// TwinCAT 3 PLC project HMI
// ProgramVersion: 3.1.4023.0
// libraries:
//   Tc2_Standard, * (Beckhoff Automation GmbH)
//   Tc2_System, * (Beckhoff Automation GmbH)
//   Tc2_Utilities, * (Beckhoff Automation GmbH)
//   Tc3_Database, * (Beckhoff Automation GmbH)
//   Tc3_Module, * (Beckhoff Automation GmbH)
// project tree:
//   DUTs/Bundle and Material/ BasicBundle.TcDUT, Bundle.TcDUT, Interval.TcDUT, Material.TcDUT, PositionMaterials.TcDUT
//   DUTs/Enums/ DatabaseStep.TcDUT, MaterialType.TcDUT
//   DUTs/ FB_TcpBlock.TcPOU, ST_TcpStructure.TcDUT
//   DUTs/String Builder/ StringBuilder.TcPOU
//   GVLs/ GVL.TcGVL
//   / PlcTask.TcTTO
//   POUs/Helper Functions/ GetMasterLength.TcPOU, GetMaterialLength.TcPOU, IntervalIsvalid.TcPOU, MetricMaterialDimensions.TcPOU, PositionIsValid.TcPOU
//   POUs/ MAIN.TcPOU, FindBundlesFromDB.TcPOU, RecalibrateRecipe.TcPOU, SqlDbReadWrite.TcPOU
// (motion and I/O tree: see PLC project dispatch)
// real-time tasks:
//   TASK PlcTask: cycle T#10ms, priority 20, ADS port 350
//   TASK PlcTask1: cycle T#10ms, priority 21, ADS port 351

CONFIGURATION HMI
    RESOURCE PLC ON TwinCAT3
        TASK PlcTask(INTERVAL := T#10ms, PRIORITY := 21);
        PROGRAM MAIN WITH PlcTask : MAIN;
    END_RESOURCE
END_CONFIGURATION

// ---- DUTs/Bundle and Material/BasicBundle.TcDUT
TYPE BasicBundle :
STRUCT
	id : STRING;
	
	weight : REAL;
	
	length : USINT;
	width : USINT;
	height : USINT;
	
	extrusionWeight : REAL;
	extrusionWidth : USINT;
	extrusionHeight : USINT;
	
	pieces : USINT;
	layers : USINT;
	piecesPerLayer : USINT;
END_STRUCT
END_TYPE

(*
barebones structure for essential bundle data that can be displayed on the HMI
refer to full structure for full recipe
*)

// ---- DUTs/Bundle and Material/Bundle.TcDUT
{attribute 'enable_dynamic_creation'}
TYPE Bundle :
STRUCT
	id : STRING;
	
	weight : REAL;
	length : USINT;
	width : USINT;
	height : USINT;
	
	pieces : USINT;
	layers : USINT;
	piecesPerLayer : USINT;
	
	extrusionWeight : REAL;
	extrusionHeight : USINT;
	extrusionWidth : USINT;
	
	processes : (AUTO_RE, AUTO_SS, MAN_RE, MAN_SS);
	reqProcesses : ARRAY[0..3] OF BOOL;
	
	coverPaper : ARRAY[0..1] OF BOOL;
	coverCardboard : ARRAY[0..1] OF BOOL;
	
	paperTop : ARRAY[0..GVL.maxPairs] OF Interval;
	paperLeft : ARRAY[0..GVL.maxPairs] OF Interval;
	paperRight : ARRAY[0..GVL.maxPairs] OF Interval;
	paperBottom : ARRAY[0..GVL.maxPairs] OF Interval;
		
	cardboard : ARRAY[0..GVL.maxPairs] OF PositionMaterials;
	cornerGuard : ARRAY[0..GVL.maxPairs] OF PositionMaterials;
	
	combinedCardboardCornerGuard : ARRAY[0..(GVL.maxPairs*2)] OF PositionMaterials;
	
	chipboard : ARRAY[0..GVL.maxPairs] OF PositionMaterials;
	woodBunk : ARRAY[0..GVL.maxPairs] OF PositionMaterials;
	
	cardboard_over_cornerGuard : BOOL;
	
	currStep : USINT; //for runtime use only
	
	//for production log database
	timeStart : TIMESTRUCT;
	timeDone : TIMESTRUCT;
END_STRUCT
END_TYPE

// ---- DUTs/Bundle and Material/Interval.TcDUT
TYPE Interval :
STRUCT
	startPos : REAL;
	endPos : REAL;
END_STRUCT
END_TYPE

// ---- DUTs/Bundle and Material/Material.TcDUT
TYPE Material :
STRUCT
	code : STRING;
	width : REAL;
	length : REAL;
	
	widthMM : INT;
	lengthMM : INT;
END_STRUCT
END_TYPE
(*
use this struct to keep track of where materials are
materials enter the system when pulled from their magazine/skid and exit the system when placed on the bundle or otherwise lost
*)

// ---- DUTs/Bundle and Material/PositionMaterials.TcDUT
TYPE PositionMaterials :
STRUCT
	position : REAL := GVL.nullPos; //default value is set to predefined constant if bundle needs less than 32 position material pairs
	
	top : STRING;
	left : STRING;
	right : STRING;
	bottom : STRING;
	
	topLeft : STRING;
	topLeftFold : USINT;
	
	topRight : STRING;
	topRightFold : USINT;
	
	bottomLeft : STRING;
	bottomLeftFold : USINT;
	
	bottomRight : STRING;
	bottomRightFold : USINT;

	wrapPoints : USINT;
	wrapRotations : USINT;
END_STRUCT
END_TYPE

// ---- DUTs/Enums/DatabaseStep.TcDUT
{attribute 'qualified_only'}
{attribute 'strict'}
TYPE DatabaseStep :
(
	RESET,
	DISCONNECT, 
	CONNECT, 
	IDLE, 
	EXECUTE, 
	LOAD_DATA,
	
	size
);
END_TYPE

// ---- DUTs/Enums/MaterialType.TcDUT
{attribute 'qualified_only'}
{attribute 'strict'}
{attribute 'to_string'}
TYPE MaterialType :
(
	PAPER,
	CARDBOARD,
	CORNER_GUARD,
	CHIPBOARD,
	WOOD_BUNK
);
END_TYPE

// ---- DUTs/ST_TcpStructure.TcDUT
TYPE ST_TcpStructure :
STRUCT
	transmissionTime : TIMESTRUCT;
	dataType : (NO_DATA, BUNDLE_TRANSFER, BUNDLE_ETA, GENERAL_EVENT)INT;
	timestamp : TIMESTRUCT;
	binaryData : ARRAY[0..50000] OF BYTE;
	jsonData : STRING(2000);
	xmlData : STRING(2000);
END_STRUCT
END_TYPE

// ---- GVLs/GVL.TcGVL
{attribute 'qualified_only'}
VAR_GLOBAL CONSTANT
	maxPairs : USINT := 16;
	initArraySize : USINT := 4;
	
	nullPos : REAL := -1;
	
	numMaterials : INT := 32;
	allMaterials : ARRAY[0..numMaterials] OF Material := [
		(code := 'PAP28', width := 28, length := -1),
		
		(code := 'CAR20S', width := 20, length := 30),
		(code := 'CAR20M', width := 20, length := 45),
		(code := 'CAR20L', width := 20, length := 60),
		(code := 'CAR28S', width := 28, length := 30),
		(code := 'CAR28M', width := 28, length := 45),
		(code := 'CAR28L', width := 28, length := 60),
		
		(code := 'COR48', width := 1.5, length := 48),
		(code := 'COR96', width := 1.5, length := 96),
		
		(code := 'CIP18', width := 20, length := 18),
		(code := 'CIP54', width := 20, length := 54),
		
		(code := 'WDT20', width := 20, length := 2.5),
		(code := 'WDT22', width := 22, length := 2.5),
		(code := 'WDT28', width := 28, length := 2.5),
		
		(code := 'WDB20', width := 20, length := 2.5),
		(code := 'WDB22', width := 22, length := 2.5),
		(code := 'WDB28', width := 28, length := 2.5),
		
		(code := 'WDS08', width := 8, length := 2.5),
		(code := 'WDS10', width := 10, length := 2.5),
		(code := 'WDS12', width := 12, length := 2.5),
		(code := 'WDS14', width := 14, length := 2.5),
		(code := 'WDS8x8', width := 16, length := 2.5),
		(code := 'WDS8x10', width := 18, length := 2.5),
		(code := 'WDS20', width := 20, length := 2.5),
		(code := 'WDS22', width := 22, length := 2.5),
		(code := 'WDS12x12', width := 24, length := 2.5),
		(code := 'WDS12x14', width := 26, length := 2.5),
		(code := 'WDS28', width := 28, length := 2.5),
		(code := 'WDS20x10', width := 30, length := 2.5),
		(code := 'WDS20x12', width := 32, length := 2.5),
		
		(code := 'WDW20', width := 20, length := 6),
		(code := 'WDW22', width := 22, length := 6)]; //+1 null material
		
	cipBuffer : INT := 2; //2in or 50mm
END_VAR
VAR_GLOBAL
	AmsNetId : T_AmsNetId;
	systemTime : TIMESTRUCT;
	
	originalBundle : Bundle; //this one stays internal
	confirmedBundle : Bundle; //this oen is editable by the HMI
END_VAR

// ---- POUs/MAIN.TcPOU
PROGRAM MAIN
VAR
	getLocalAmsNetId : FB_GetLocalAmsNetId;
	getLocalSystemTime : FB_LocalSystemTime;
	
	id : STRING;
	queryId : STRING;
	stringBuilder : StringBuilder;
	
	original : Bundle;
	confirmed : Bundle;
END_VAR
VAR CONSTANT
	AUTO_RE : INT := 0;
	AUTO_SS : INT := 1;
	MAN_RE : INT := 2;
	MAN_SS : INT := 3;
END_VAR

getLocalSystemTime(
	sNetID:= GVL.AmsNetId, 
	bEnable:= TRUE, 
	dwCycle:= 1, 
	dwOpt:= , 
	tTimeout:= , 
	bValid=> , 
	systemTime=> GVL.systemTime, 
	tzID=> );

IF NOT setup() THEN
	RETURN;
END_IF

MetricMaterialDimensions(GVL.allMaterials);

queryId := stringBuilder
	.concatWith('%')
	.concatWith(id)
	.concatWith('%')
	.getResult();
stringBuilder.reset();

FindBundlesFromDB(id := queryId);

IF confirmed.length <> original.length THEN
	RecalibrateRecipe(original := original, confirmed := confirmed);
	
	IF RecalibrateRecipe.reject THEN //send to manual processes
		confirmed.reqProcesses[AUTO_RE] := FALSE;
		confirmed.reqProcesses[AUTO_SS] := FALSE;
		confirmed.reqProcesses[MAN_RE] := TRUE;
		confirmed.reqProcesses[MAN_SS] := TRUE;	
	END_IF
ELSE
	//use as is
END_IF

METHOD setup : BOOL
VAR_INPUT
END_VAR
getLocalAmsNetId(
	bExecute:= TRUE, 
	tTimeOut:= T#1S, 
	bBusy=> , 
	bError=> , 
	nErrId=> , 
	AddrString=> GVL.AmsNetId, 
	AddrBytes=> );

getLocalAmsNetId.bExecute := FALSE;

setup := (GVL.AmsNetId <> '' AND GVL.AmsNetId <> '0.0.0.0.0.0');
END_METHOD

END_PROGRAM

// ---- DUTs/String Builder/StringBuilder.TcPOU
FUNCTION_BLOCK StringBuilder
VAR
	result : STRING(1000);
END_VAR

METHOD concatStringArray : STRING(1000)
VAR_IN_OUT
	arr : ARRAY[*] OF STRING;
END_VAR
VAR
	temp : STRING(1000);
END_VAR
END_METHOD

METHOD concatWith : REFERENCE TO StringBuilder
VAR_INPUT
	target : STRING;
END_VAR
CONCAT2(ADR(result), ADR(target), ADR(result), SIZEOF(result));
concatWith REF= THIS^;
END_METHOD

METHOD getResult : STRING(1000)
getResult := result;
END_METHOD

METHOD reset : BOOL
VAR_INPUT
END_VAR
result := '';
END_METHOD

END_FUNCTION_BLOCK

// ---- POUs/Helper Functions/MetricMaterialDimensions.TcPOU
FUNCTION MetricMaterialDimensions : BOOL
VAR_IN_OUT
	materials : ARRAY[*] OF Material;
END_VAR
VAR
	i : DINT;
END_VAR

FOR i:=LOWER_BOUND(materials, 1) TO UPPER_BOUND(materials, 1) BY 1 DO
	materials[i].lengthMM := TO_INT(materials[i].length * 25.4);
	materials[i].widthMM := TO_INT(materials[i].width * 25.4);
END_FOR

END_FUNCTION

// ---- POUs/FindBundlesFromDB.TcPOU
PROGRAM FindBundlesFromDB EXTENDS SqldbReadWrite
VAR_INPUT
	id : STRING;
END_VAR
VAR_OUTPUT
	basicBundlesArr : ARRAY[0..20-1] OF BasicBundle;
END_VAR
VAR
	fbSQLCommand : FB_SQLCommandEvt(sNetID := '', tTimeout := T#5S);
	fbSQLDatabase : FB_SQLDatabaseEvt (sNetID := '', tTimeout := T#5S);
	fbSQLResult : FB_SQLResultEvt(sNetID:='', tTimeout:=T#5S);
	
	query : STRING(1000);
	//step : (RESET, CONNECT, IDLE, EXECUTE, LOAD_DATA, DISCONNECT);
END_VAR
VAR
	stringBuilder : StringBuilder;
	i : INT;
END_VAR

IF NOT ready THEN
	setup();
	RETURN;
END_IF

CASE step OF
	(*
	RESET:
		step := DISCONNECT;
		
	CONNECT:
		IF fbSQLDatabase.Connect(1) THEN
			IF NOT fbSqlDatabase.bError THEN
				step := IDLE;
			END_IF
		END_IF
	*)
	IDLE:
		IF fbSQLDatabase.CreateCmd(ADR(fbSQLCommand)) THEN
			step := EXECUTE;
		END_IF
	
	EXECUTE:
		createQuery();
		IF fbSQLCommand.ExecuteDataReturn(ADR(query), SIZEOF(query), ADR(fbSqlResult)) THEN
			step := IDLE;
		END_IF
	
	LOAD_DATA:
		(*
		fbSqlResult.Read(0, 1, ADR(existingID), SIZEOF(existingID), TRUE, FALSE);
		IF BundleData.id = existingID THEN
			bundleExists := TRUE;
		ELSE
			bundleExists := FALSE;
		END_IF
		IF fbSQLDatabase.Disconnect() THEN
			fbSqlResult.Release();
			checkExistingBundles := TRUE;
			dbCheckStep := CONNECT;
		END_IF
		*)
		
	DISCONNECT:
		IF fbSQLDatabase.Disconnect() THEN
			step := CONNECT;
		END_IF
END_CASE

METHOD PRIVATE createQuery : BOOL
IF id = '' THEN //FINISH WITH OTHER BASIC ATTRIBUTES
	CONCAT2(ADR(query), ADR('SELECT BundleID FROM "Bundle Data - Prototype"'), ADR(query), SIZEOF(query));
ELSE
	CONCAT2(ADR(query), ADR('SELECT BundleID FROM "Bundle Data - Prototype" WHERE BundleID = $''), ADR(query), SIZEOF(query));
	CONCAT2(ADR(query), ADR(id), ADR(query), SIZEOF(query));
	CONCAT2(ADR(query), ADR('$''), ADR(query), SIZEOF(query));
END_IF

createQuery := TRUE;
END_METHOD

METHOD queryBasicAttributes : BOOL
VAR_INPUT
END_VAR
END_METHOD

METHOD queryPackagingRecipe : BOOL
VAR_INPUT
	material : MaterialType;
END_VAR
VAR
	sMaterial : STRING;
END_VAR
sMaterial := TO_STRING(material);

IF i >= GVL.maxPairs THEN
	i := 0;
END_IF

sMaterial := stringBuilder
	.concatWith(
		'SELECT
		(position, top, sides, bottom, upperCorners, upperCorners_foldRatio, lowerCorners, lowerCorners_foldRatio)
		FROM ______ 
		WHERE (')
		
	.concatWith('bundleID = ')
	.concatWith('$'')
	.concatWith(TO_STRING(id))
	.concatWith('$'')
	
	.concatWith(' AND ')
	
	.concatWith('arrayIndex = ')
	.concatWith(TO_STRING(i))
	.concatWith(')')
	.getResult();
(*

FOR i:=0 TO 16 BY 1 DO


select (position, top, sides, bottom, upperCorners, upperCorners_foldRatio, lowerCorners, lowerCorners_foldRatio) from 
where (bundleID = bundle.id and arrayIndex = 1)

//copy the resulting cache into a bundle.<material>[i] (a PositionMaterial struct)
//do this for all material arrays


END_FORR

*)
END_METHOD

METHOD setup : BOOL
CASE step OF
	RESET:
		step := DISCONNECT;
		
	CONNECT:
		IF fbSQLDatabase.Connect(1) THEN
			IF NOT fbSqlDatabase.bError THEN
				step := IDLE;
				setup := TRUE;
			END_IF
		END_IF
		
	DISCONNECT:
		IF fbSQLDatabase.Disconnect() THEN
			step := CONNECT;
		END_IF
END_CASE
END_METHOD

END_PROGRAM

// ---- POUs/SqlDbReadWrite.TcPOU
PROGRAM SqlDbReadWrite
VAR_OUTPUT
	ready : BOOL;
END_VAR
VAR
	fbSQLCommand : FB_SQLCommandEvt(sNetID := '', tTimeout := T#5S);
	fbSQLDatabase : FB_SQLDatabaseEvt (sNetID := '', tTimeout := T#5S);
	fbSQLResult : FB_SQLResultEvt(sNetID:='', tTimeout:=T#5S);
	
	query : STRING(1000);
	step : DatabaseStep;
	
	cachedBuffer : ARRAY[0..100000] OF BYTE;
END_VAR

IF NOT ready THEN
	setup();
	RETURN;
END_IF

CASE step OF
	DatabaseStep.IDLE:
		IF fbSQLDatabase.CreateCmd(ADR(fbSQLCommand)) THEN
			step := DatabaseStep.EXECUTE;
		END_IF
		
	DatabaseStep.EXECUTE:
		IF fbSQLCommand.ExecuteDataReturn(ADR(query), SIZEOF(query), ADR(fbSqlResult)) THEN
			query := '';
			step := DatabaseStep.LOAD_DATA;
		END_IF
		
	DatabaseStep.LOAD_DATA:
		fbSqlResult.Read(
			nStartIndex := 0,
			nRecordCount := 1,
			pData := ADR(cachedBuffer),
			cbData := SIZEOF(cachedBuffer),
			bWithVerifying := FALSE,
			bDataRelease := FALSE);
			
END_CASE

METHOD execute : BOOL
VAR_INPUT
	queryInstruction : STRING(1000);
END_VAR
query := queryInstruction;
END_METHOD

METHOD reset : BOOL
VAR_INPUT
END_VAR
step := RESET;
END_METHOD

METHOD setup : BOOL
CASE step OF
	DatabaseStep.RESET:
		step := DatabaseStep.DISCONNECT;
		
	DatabaseStep.CONNECT:
		IF fbSQLDatabase.Connect(1) THEN
			IF NOT fbSqlDatabase.bError THEN
				step := DatabaseStep.IDLE;
				setup := TRUE;
			END_IF
		END_IF
		
	DatabaseStep.DISCONNECT:
		IF fbSQLDatabase.Disconnect() THEN
			step := DatabaseStep.CONNECT;
		END_IF
END_CASE
END_METHOD

END_PROGRAM

// ---- POUs/RecalibrateRecipe.TcPOU
PROGRAM RecalibrateRecipe
VAR_INPUT
	original : REFERENCE TO Bundle;
	confirmed : REFERENCE TO Bundle;
END_VAR
VAR
	lengthDifference : REAL;
	minAllowableLength : REAL;
	lengthShortenedDifferenceMax : REAL;
	
	lengthDifferenceFactor : REAL;
	
	cipLength : REAL;
	
	i : INT;
END_VAR
VAR_OUTPUT
	reject : BOOL;
END_VAR

//original REF= GVL.originalBundle;
//confirmed REF= GVL.confirmedBundle;

lengthDifference := confirmed.length - original.length;
minAllowableLength := cipLength + (2 * GVL.cipBuffer);
lengthShortenedDifferenceMax := original.length - minAllowableLength;

lengthDifferenceFactor := confirmed.length/original.length;

reject := FALSE; //reset rejection status
IF confirmed.length < original.length THEN	
	calibrate(confirmed.chipboard);
	calibrate(confirmed.cornerGuard);
	optimize(confirmed.cardboard);
	//optimize(confirmed.paperTop);
ELSIF confirmed.length > original.length THEN
	(*
	split the bundle in half
	keep all materials at the same distance from the closer edge (front/back)
	or
	//THIS
	keep first and last material in place
	scale the position of everything else in the middle
	*)
	scale(confirmed.cardboard);
	scale(confirmed.cornerGuard);
	scale(confirmed.chipboard);
END_IF

METHOD calibrate : BOOL
VAR_IN_OUT
	pairsArr : ARRAY[*] OF PositionMaterials;
END_VAR
VAR
	currPair : REFERENCE TO PositionMaterials;
	prevPair : REFERENCE TO PositionMaterials;
	
	accumulatedGaps : REAL;
	currMaterialFrontPos : REAL;
	prevMaterialBackPos : REAL;	
	currGap : REAL;
	
	tempReject : BOOL;
END_VAR
(*
this method is for materials that cannot overlap and have strict acceptance/rejection criteria
currently only used by cornerboard and chipboard
*)
cipLength := 0;

FOR i:=0 TO GVL.maxPairs BY 1 DO
	currPair REF= pairsArr[i];
	IF currPair.position = GVL.nullPos THEN
		CONTINUE;
	END_IF
	
	cipLength := cipLength + GetMasterLength(currPair);
END_FOR

IF confirmed.length < minAllowableLength THEN
	tempReject := TRUE;
	RETURN;
END_IF //guard clause

FOR i:=1 TO GVL.maxPairs BY 1 DO
	currPair REF= pairsArr[i];
	prevPair REF= pairsArr[i-1];
	
	IF currPair.position = GVL.nullPos THEN
		CONTINUE;
	END_IF
	
	
	currMaterialFrontPos := currPair.position - GetMasterLength(currPair)/2; //- front, + back
	prevMaterialBackPos := prevPair.position + GetMasterLength(prevPair)/2;
	
	currGap := currMaterialFrontPos - prevMaterialBackPos;
	
	currPair.position := currPair.position - (((1 - lengthDifference/lengthShortenedDifferenceMax) * currGap) - accumulatedGaps);
	accumulatedGaps := accumulatedGaps + currGap;
END_FOR
tempReject := FALSE;

reject := MAX(reject, tempReject);
END_METHOD

METHOD chipboard : BOOL
VAR
	currPair : REFERENCE TO PositionMaterials;
	prevPair : REFERENCE TO PositionMaterials;
	
	accumulatedGaps : REAL;
	currMaterialFrontPos : REAL;
	prevMaterialBackPos : REAL;	
	currGap : REAL;
END_VAR
cipLength := 0;

FOR i:=0 TO GVL.maxPairs BY 1 DO
	currPair REF= confirmed.chipboard[i];
	IF currPair.position = GVL.nullPos THEN
		CONTINUE;
	END_IF
	
	cipLength := cipLength + GetMasterLength(currPair);
END_FOR

IF confirmed.length < minAllowableLength THEN
	reject := TRUE;
	RETURN;
END_IF //guard clause

FOR i:=1 TO GVL.maxPairs BY 1 DO
	currPair REF= confirmed.chipboard[i];
	prevPair REF= confirmed.chipboard[i-1];
	
	IF currPair.position = GVL.nullPos THEN
		CONTINUE;
	END_IF
	
	
	currMaterialFrontPos := currPair.position - GetMasterLength(currPair)/2; //- front, + back
	prevMaterialBackPos := prevPair.position + GetMasterLength(prevPair)/2;
	
	currGap := currMaterialFrontPos - prevMaterialBackPos;
	
	currPair.position := currPair.position - (((1 - lengthDifference/lengthShortenedDifferenceMax) * currGap) - accumulatedGaps);
	accumulatedGaps := accumulatedGaps + currGap;
END_FOR
reject := FALSE;
END_METHOD

METHOD cornerboard : BOOL
VAR
	currPair : REFERENCE TO PositionMaterials;
	prevPair : REFERENCE TO PositionMaterials;
	
	accumulatedGaps : REAL;
	currMaterialFrontPos : REAL;
	prevMaterialBackPos : REAL;	
	currGap : REAL;
	i : BOOL;
END_VAR
END_METHOD

METHOD optimize : BOOL
VAR_IN_OUT
	pairsArr : ARRAY[*] OF PositionMaterials;
END_VAR
VAR
	currPair : REFERENCE TO PositionMaterials;
	prevPair : REFERENCE TO PositionMaterials;
	
	accumulatedGaps : REAL;
	currMaterialFrontPos : REAL;
	prevMaterialBackPos : REAL;	
	currGap : REAL;
	
	tempReject : BOOL;
END_VAR
(*
this method is for materials are allowed to overlap
acceptance/rejection conditions may be more lax
currently used by paper, cardboard
*)
END_METHOD

METHOD scale : BOOL
VAR_IN_OUT
	pairsArr : ARRAY[*] OF PositionMaterials;
END_VAR
VAR
	currPair : REFERENCE TO PositionMaterials;
	firstPair : REFERENCE TO PositionMaterials;
	lastPair : REFERENCE TO PositionMaterials;
	firstPairIndex : INT;
	lastPairIndex : INT;
	
	lastPairLength : REAL;
END_VAR
FOR i:=0 TO GVL.maxPairs BY 1 DO //find first and last pair
	currPair REF= pairsArr[i];
	
	IF PositionIsValid(currPair) THEN
		IF NOT __ISVALIDREF(firstPair) THEN //set first pair once only
			firstPair REF= pairsArr[i];
			firstPairIndex := i;
		END_IF
		lastPair REF= pairsArr[i]; //keep setting last pair
		lastPairIndex := i;
	END_IF
END_FOR

FOR i:=firstPairIndex+1 TO lastPairIndex-1 BY 1 DO
	pairsArr[i].position := pairsArr[i].position * lengthDifferenceFactor;
END_FOR

//leave first pair untouched, recalculate last pair position
lastPair.position := confirmed.length - GetMasterLength(lastPair)/2;
END_METHOD

METHOD scalePaper : BOOL
VAR_IN_OUT
	paperArr : ARRAY[*] OF Interval;
END_VAR
VAR
	currPair : REFERENCE TO Interval;
	firstPair : REFERENCE TO Interval;
	lastPair : REFERENCE TO Interval;
	firstPairIndex : INT;
	lastPairIndex : INT;
	
	lastPairEnd : REAL;
END_VAR
FOR i:=0 TO GVL.maxPairs BY 1 DO //find first and last pair
	currPair REF= paperArr[i];
	
	IF IntervalIsValid(currPair) THEN
		IF NOT __ISVALIDREF(firstPair) THEN //set first pair once only
			firstPair REF= paperArr[i];
			firstPairIndex := i;
		END_IF
		lastPair REF= paperArr[i]; //keep setting last pair
		lastPairIndex := i;
	END_IF
END_FOR

FOR i:=firstPairIndex+1 TO lastPairIndex-1 BY 1 DO
	paperArr[i].startPos := paperArr[i].startPos * lengthDifferenceFactor;
	paperArr[i].endPos := paperArr[i].endPos * lengthDifferenceFactor;
END_FOR

//leave first pair start pos
firstPair.endPos := firstPair.endPos * lengthDifferenceFactor;

lastPair.startPos := lastPair.startPos * lengthDifferenceFactor;
//leave last pair end pos
END_METHOD

END_PROGRAM

// ---- POUs/Helper Functions/GetMasterLength.TcPOU
FUNCTION GetMasterLength : REAL
VAR_INPUT
	currentPair : REFERENCE TO PositionMaterials;
END_VAR
VAR
	topLength : REAL;
	leftLength : REAL;
	rightLength : REAL;
	bottomLength : REAL;
	
	topLeftLength : REAL;
	topRightLength : REAL;
	bottomLeftLength : REAL;
	bottomRightLength : REAL;
END_VAR

topLength := GetMaterialLength(currentPair.top);
leftLength := GetMaterialLength(currentPair.left);
rightLength := GetMaterialLength(currentPair.right);
bottomLength := GetMaterialLength(currentPair.bottom);

topLeftLength := GetMaterialLength(currentPair.topLeft);
topRightLength := GetMaterialLength(currentPair.topRight);
bottomLeftLength := GetMaterialLength(currentPair.bottomLeft);
bottomRightLength := GetMaterialLength(currentPair.bottomRight);

GetMasterLength := MAX(topLength, leftLength, rightLength, bottomLength, topLeftLength, topRightLength, bottomLeftLength, bottomRightLength);

END_FUNCTION

// ---- POUs/Helper Functions/GetMaterialLength.TcPOU
FUNCTION GetMaterialLength : REAL
VAR_INPUT
	material : STRING;
END_VAR
VAR
	i : INT;
END_VAR

FOR i:=0 TO GVL.numMaterials BY 1 DO
	IF GVL.allMaterials[i].code = material THEN
		getMaterialLength := GVL.allMaterials[i].length;
		RETURN;
	END_IF
END_FOR
//otherwise, return 0
//GetMaterialLength := 0;

END_FUNCTION

// ---- POUs/Helper Functions/PositionIsValid.TcPOU
FUNCTION PositionIsValid : BOOL
VAR_INPUT
	pair : REFERENCE TO PositionMaterials;
END_VAR

PositionIsValid := (
	pair.position <> GVL.nullPos AND
	(
		pair.top <> '' OR
		pair.left <> '' OR
		pair.right <> '' OR
		pair.bottom <> '' OR
		
		pair.topLeft <> '' OR
		pair.topRight <> '' OR
		pair.bottomLeft <> '' OR
		pair.bottomRight <> ''
	));

END_FUNCTION

// ---- POUs/Helper Functions/IntervalIsvalid.TcPOU
FUNCTION IntervalIsvalid : BOOL
VAR_INPUT
	pair : REFERENCE TO Interval;
END_VAR

IntervalIsValid := (
	pair.startPos <> GVL.nullPos AND 
	pair.endPos <> GVL.nullPos AND 
	pair.startPos < pair.endPos);

END_FUNCTION

// ---- DUTs/FB_TcpBlock.TcPOU
FUNCTION_BLOCK FB_TcpBlock
VAR
	tcpTime : TIMESTRUCT;
	
	dataType : (NO_DATA, BUNDLE_TRANSFER, BUNDLE_ETA, GENERAL_EVENT);
	timestamp : TIMESTRUCT;
	
	binaryData : ARRAY[0..50000] OF BYTE;
	jsonData : STRING(2000);
	xmlData : STRING(2000);
END_VAR

METHOD sendBundleETA : BOOL
VAR_INPUT
	eta : TIMESTRUCT;
	bundleId : STRING;
END_VAR
END_METHOD

METHOD sendBundleTransfer : BOOL
VAR_INPUT
END_VAR
END_METHOD

METHOD setTcpTime : BOOL
tcpTime := GVL.systemTime;
END_METHOD

END_FUNCTION_BLOCK
